(* PLC project Unnamed, Unknown Unnamed 1 *)
(* stored: creationDateTime 2023-03-28T20:41:08, modificationDateTime 2023-04-03T10:58:40 *)

PROGRAM FactoryIO
  VAR
    Stop_Button AT %IX100.0 : BOOL;
    Start_Button AT %IX100.1 : BOOL;
    Conveyor AT %QX100.0 : BOOL;
  END_VAR

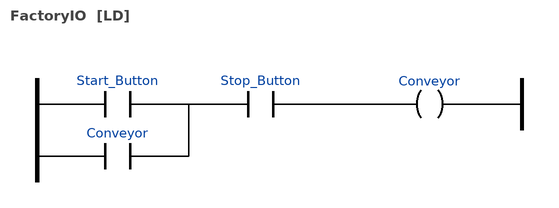
(* LD diagram, written out as Structured Text *)
Conveyor := (Start_Button OR Conveyor) AND Stop_Button;
END_PROGRAM

CONFIGURATION Config0
  RESOURCE Res0 ON PLC
    TASK task0(INTERVAL := T#20ms, PRIORITY := 0);
    PROGRAM instance0 WITH task0 : FactoryIO;
  END_RESOURCE
END_CONFIGURATION
